// TIA Portal V20 export
TYPE "LER_zp_CITI_Configuration"
// stored: Access Published
   STRUCT
      Instance : DInt;   // Map Instance
      UpdatePriority : DInt;   // Update Priority
      Features : "LER_zp_CITI_Features";   // Features
      Parameters { S7_SetPoint := 'True'} : "LER_zp_CITI_Parameters";   // Parameters
   END_STRUCT;
END_TYPE
